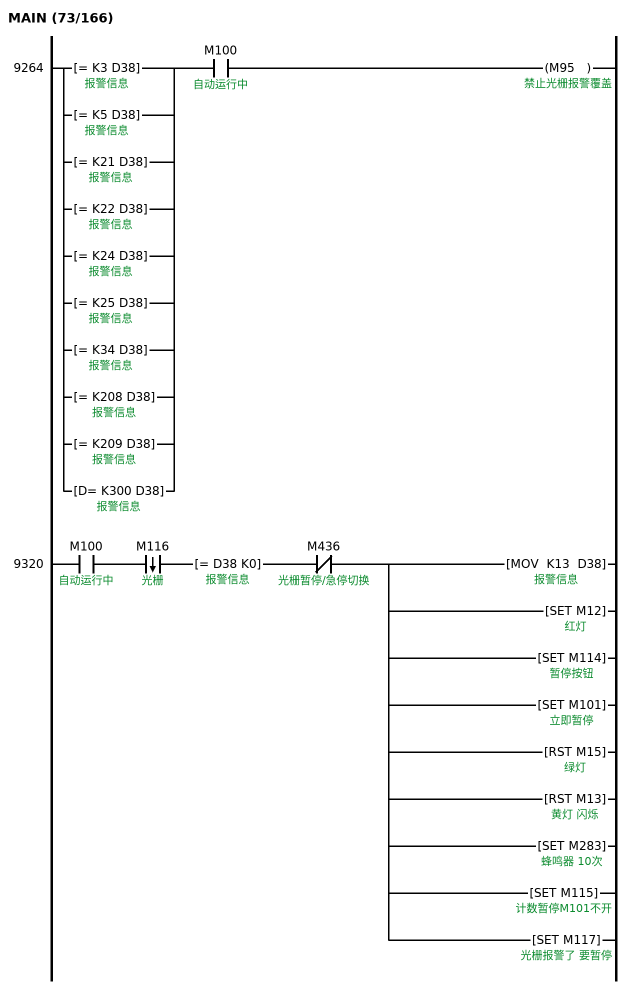
[picture p72: ladder of MAIN, rungs at steps 9264 to 9320]
9264  LD=     K3 D38  ; 报警信息
      OR=     K5 D38  ; 报警信息
      OR=     K21 D38  ; 报警信息
      OR=     K22 D38  ; 报警信息
      OR=     K24 D38  ; 报警信息
      OR=     K25 D38  ; 报警信息
      OR=     K34 D38  ; 报警信息
      OR=     K208 D38  ; 报警信息
      OR=     K209 D38  ; 报警信息
      ORD=    K300 D38  ; 报警信息
      AND     M100  ; 自动运行中
      OUT     M95  ; 禁止光栅报警覆盖
9320  LD      M100  ; 自动运行中
      ANDF    M116  ; 光栅
      AND=    D38 K0  ; 报警信息
      ANI     M436  ; 光栅暂停/急停切换
      MOV     K13 D38
      SET     M12  ; 红灯
      SET     M114  ; 暂停按钮
      SET     M101  ; 立即暂停
      RST     M15  ; 绿灯
      RST     M13  ; 黄灯 闪烁
      SET     M283  ; 蜂鸣器 10次
      SET     M115  ; 计数暂停M101不开
      SET     M117  ; 光栅报警了 要暂停
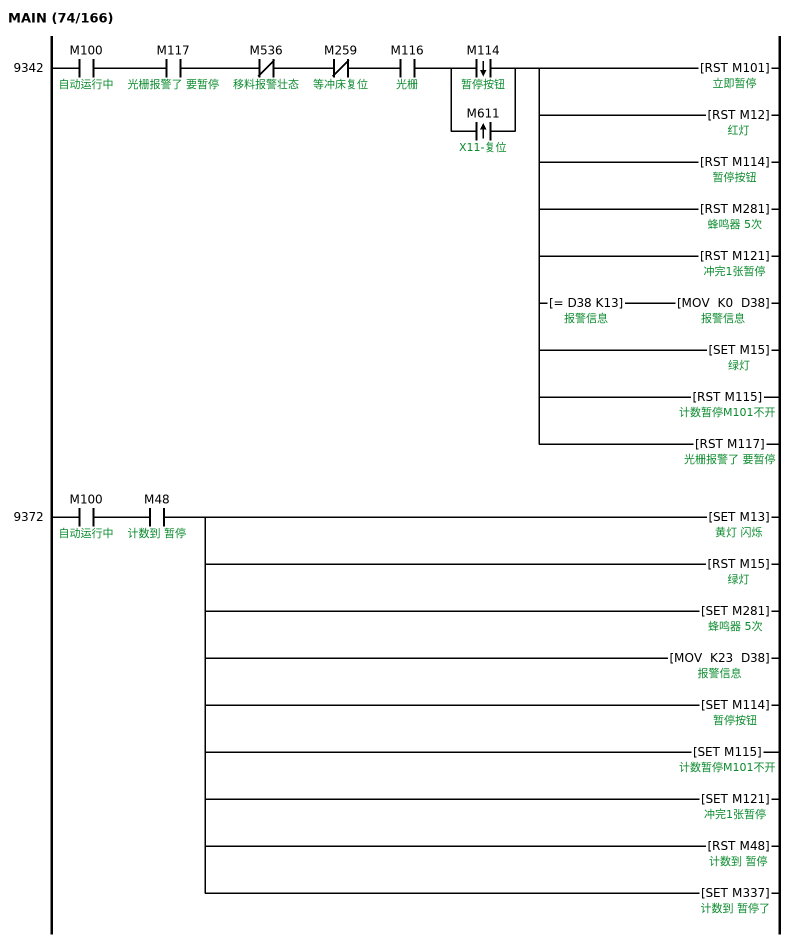
9342  LD      M100  ; 自动运行中
      AND     M117  ; 光栅报警了 要暂停
      ANI     M536  ; 移料报警壮态
      ANI     M259  ; 等冲床复位
      AND     M116  ; 光栅
      LDF     M114  ; 暂停按钮
      ORP     M611  ; X11-复位
      ANB
      RST     M101  ; 立即暂停
      RST     M12  ; 红灯
      RST     M114  ; 暂停按钮
      RST     M281  ; 蜂鸣器 5次
      RST     M121  ; 冲完1张暂停
      MPS
      AND=    D38 K13  ; 报警信息
      MOV     K0 D38
      MPP
      SET     M15  ; 绿灯
      RST     M115  ; 计数暂停M101不开
      RST     M117  ; 光栅报警了 要暂停
9372  LD      M100  ; 自动运行中
      AND     M48  ; 计数到 暂停
      SET     M13  ; 黄灯 闪烁
      RST     M15  ; 绿灯
      SET     M281  ; 蜂鸣器 5次
      MOV     K23 D38
      SET     M114  ; 暂停按钮
      SET     M115  ; 计数暂停M101不开
      SET     M121  ; 冲完1张暂停
      RST     M48  ; 计数到 暂停
      SET     M337  ; 计数到 暂停了
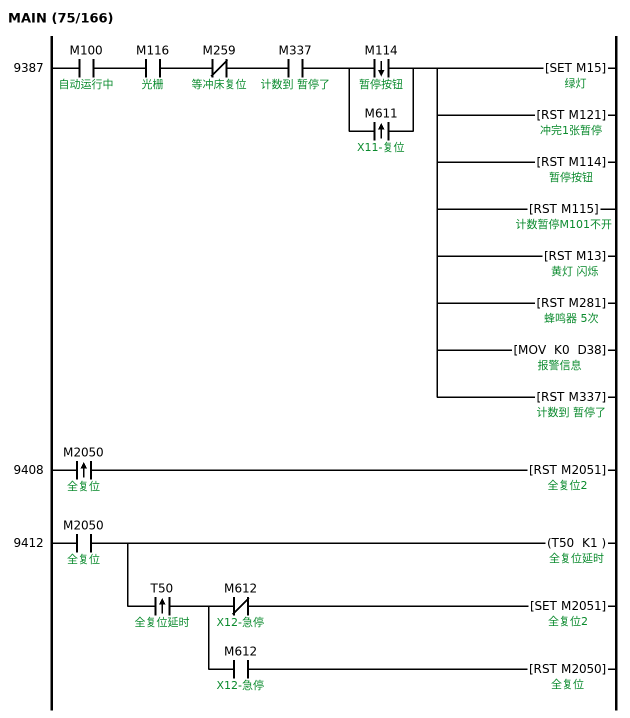
9387  LD      M100  ; 自动运行中
      AND     M116  ; 光栅
      ANI     M259  ; 等冲床复位
      AND     M337  ; 计数到 暂停了
      LDF     M114  ; 暂停按钮
      ORP     M611  ; X11-复位
      ANB
      SET     M15  ; 绿灯
      RST     M121  ; 冲完1张暂停
      RST     M114  ; 暂停按钮
      RST     M115  ; 计数暂停M101不开
      RST     M13  ; 黄灯 闪烁
      RST     M281  ; 蜂鸣器 5次
      MOV     K0 D38
      RST     M337  ; 计数到 暂停了
9408  LDP     M2050  ; 全复位
      RST     M2051  ; 全复位2
9412  LD      M2050  ; 全复位
      OUT     T50 K1  ; 全复位延时
      ANDP    T50  ; 全复位延时
      MPS
      ANI     M612  ; X12-急停
      SET     M2051  ; 全复位2
      MPP
      AND     M612  ; X12-急停
      RST     M2050  ; 全复位
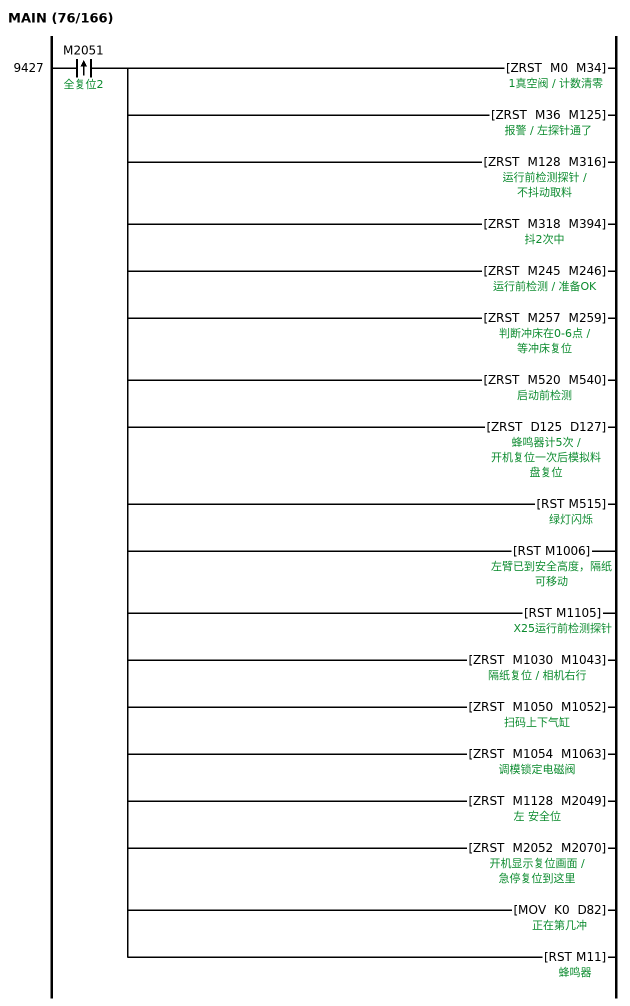
9427  LDP     M2051  ; 全复位2
      ZRST    M0 M34
      ZRST    M36 M125
      ZRST    M128 M316
      ZRST    M318 M394
      ZRST    M245 M246
      ZRST    M257 M259
      ZRST    M520 M540
      ZRST    D125 D127
      RST     M515  ; 绿灯闪烁
      RST     M1006  ; 左臂已到安全高度，隔纸可移动
      RST     M1105  ; X25运行前检测探针
      ZRST    M1030 M1043
      ZRST    M1050 M1052
      ZRST    M1054 M1063
      ZRST    M1128 M2049
      ZRST    M2052 M2070
      MOV     K0 D82
      RST     M11  ; 蜂鸣器
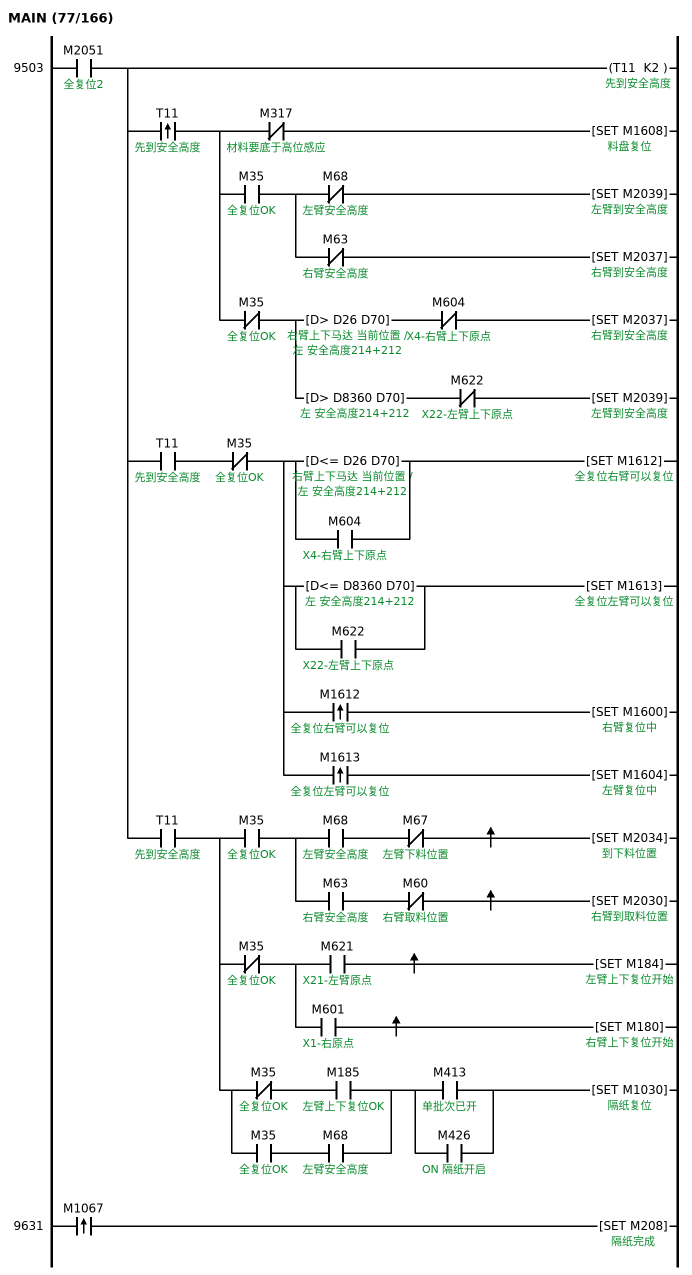
9503  LD      M2051  ; 全复位2
      OUT     T11 K2  ; 先到安全高度
      MPS
      ANDP    T11  ; 先到安全高度
      MPS
      ANI     M317  ; 材料要底于高位感应
      SET     M1608  ; 料盘复位
      MRD
      AND     M35  ; 全复位OK
      MPS
      ANI     M68  ; 左臂安全高度
      SET     M2039  ; 左臂到安全高度
      MPP
      ANI     M63  ; 右臂安全高度
      SET     M2037  ; 右臂到安全高度
      MPP
      ANI     M35  ; 全复位OK
      MPS
      ANDD>   D26 D70  ; 右臂上下马达 当前位置 / 左 安全高度214+212
      ANI     M604  ; X4-右臂上下原点
      SET     M2037  ; 右臂到安全高度
      MPP
      ANDD>   D8360 D70  ; 左 安全高度214+212
      ANI     M622  ; X22-左臂上下原点
      SET     M2039  ; 左臂到安全高度
      MRD
      AND     T11  ; 先到安全高度
      ANI     M35  ; 全复位OK
      MPS
      LDD<=   D26 D70  ; 右臂上下马达 当前位置 / 左 安全高度214+212
      OR      M604  ; X4-右臂上下原点
      ANB
      SET     M1612  ; 全复位右臂可以复位
      MRD
      LDD<=   D8360 D70  ; 左 安全高度214+212
      OR      M622  ; X22-左臂上下原点
      ANB
      SET     M1613  ; 全复位左臂可以复位
      MRD
      ANDP    M1612  ; 全复位右臂可以复位
      SET     M1600  ; 右臂复位中
      MPP
      ANDP    M1613  ; 全复位左臂可以复位
      SET     M1604  ; 左臂复位中
      MPP
      AND     T11  ; 先到安全高度
      MPS
      AND     M35  ; 全复位OK
      MPS
      AND     M68  ; 左臂安全高度
      ANI     M67  ; 左臂下料位置
      MEP
      SET     M2034  ; 到下料位置
      MPP
      AND     M63  ; 右臂安全高度
      ANI     M60  ; 右臂取料位置
      MEP
      SET     M2030  ; 右臂到取料位置
      MRD
      ANI     M35  ; 全复位OK
      MPS
      AND     M621  ; X21-左臂原点
      MEP
      SET     M184  ; 左臂上下复位开始
      MPP
      AND     M601  ; X1-右原点
      MEP
      SET     M180  ; 右臂上下复位开始
      MPP
      LDI     M35  ; 全复位OK
      AND     M185  ; 左臂上下复位OK
      LD      M35  ; 全复位OK
      AND     M68  ; 左臂安全高度
      ORB
      ANB
      LD      M413  ; 单批次已开
      OR      M426  ; ON 隔纸开启
      ANB
      SET     M1030  ; 隔纸复位
9631  LDP     M1067
      SET     M208  ; 隔纸完成
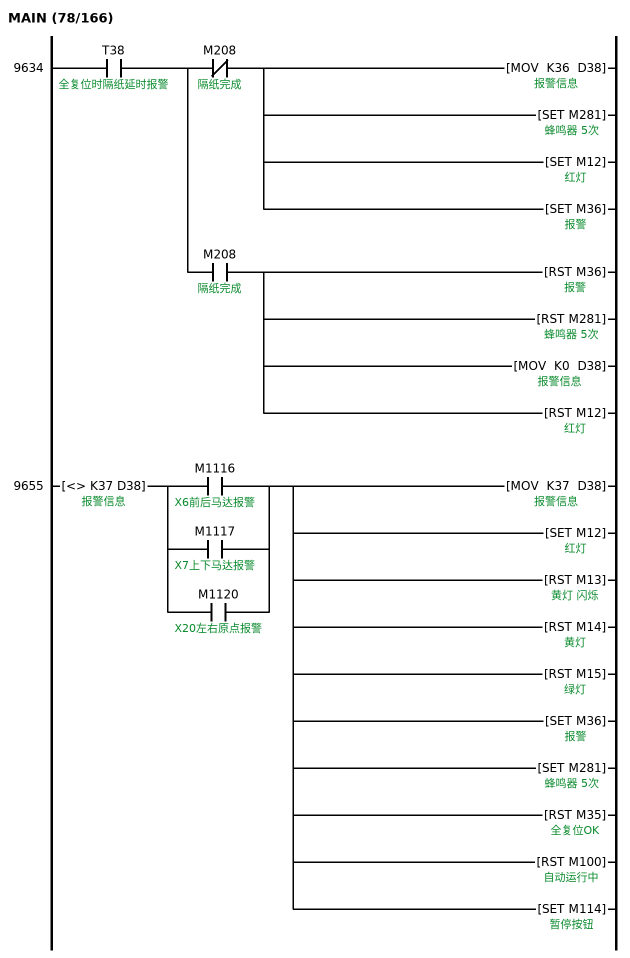
9634  LD      T38  ; 全复位时隔纸延时报警
      MPS
      ANI     M208  ; 隔纸完成
      MOV     K36 D38
      SET     M281  ; 蜂鸣器 5次
      SET     M12  ; 红灯
      SET     M36  ; 报警
      MPP
      AND     M208  ; 隔纸完成
      RST     M36  ; 报警
      RST     M281  ; 蜂鸣器 5次
      MOV     K0 D38
      RST     M12  ; 红灯
9655  LD<>    K37 D38  ; 报警信息
      LD      M1116  ; X6前后马达报警
      OR      M1117  ; X7上下马达报警
      OR      M1120  ; X20左右原点报警
      ANB
      MOV     K37 D38
      SET     M12  ; 红灯
      RST     M13  ; 黄灯 闪烁
      RST     M14  ; 黄灯
      RST     M15  ; 绿灯
      SET     M36  ; 报警
      SET     M281  ; 蜂鸣器 5次
      RST     M35  ; 全复位OK
      RST     M100  ; 自动运行中
      SET     M114  ; 暂停按钮
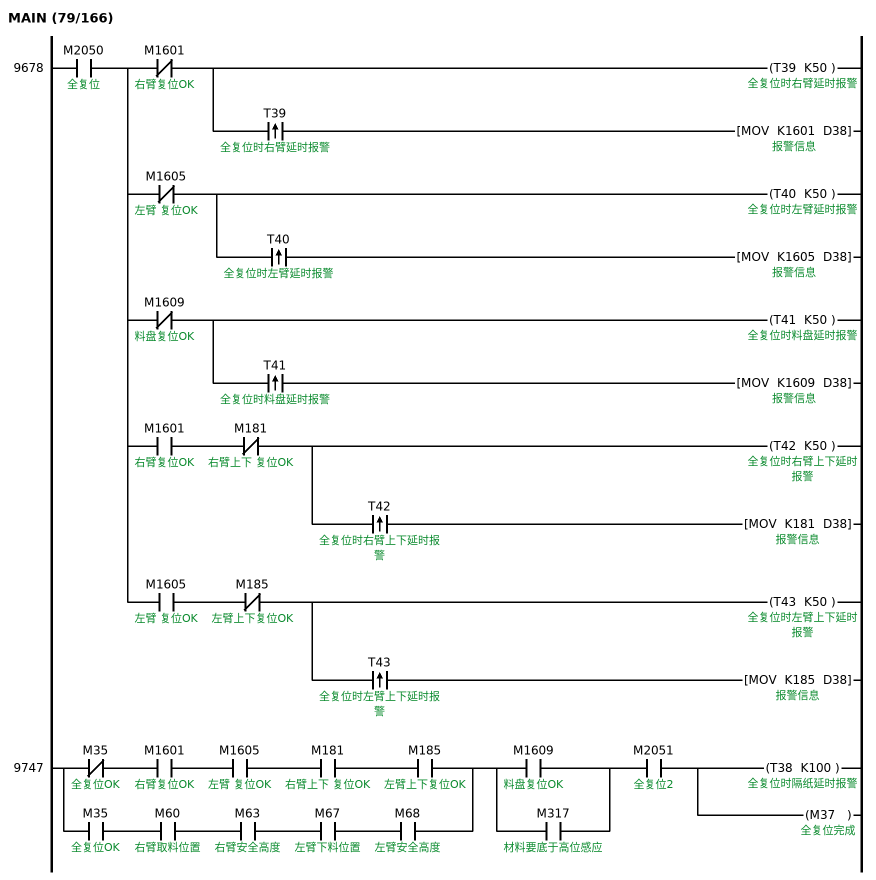
9678  LD      M2050  ; 全复位
      MPS
      ANI     M1601  ; 右臂复位OK
      OUT     T39 K50  ; 全复位时右臂延时报警
      ANDP    T39  ; 全复位时右臂延时报警
      MOV     K1601 D38
      MRD
      ANI     M1605  ; 左臂 复位OK
      OUT     T40 K50  ; 全复位时左臂延时报警
      ANDP    T40  ; 全复位时左臂延时报警
      MOV     K1605 D38
      MRD
      ANI     M1609  ; 料盘复位OK
      OUT     T41 K50  ; 全复位时料盘延时报警
      ANDP    T41  ; 全复位时料盘延时报警
      MOV     K1609 D38
      MRD
      AND     M1601  ; 右臂复位OK
      ANI     M181  ; 右臂上下 复位OK
      OUT     T42 K50  ; 全复位时右臂上下延时报警
      ANDP    T42  ; 全复位时右臂上下延时报警
      MOV     K181 D38
      MPP
      AND     M1605  ; 左臂 复位OK
      ANI     M185  ; 左臂上下复位OK
      OUT     T43 K50  ; 全复位时左臂上下延时报警
      ANDP    T43  ; 全复位时左臂上下延时报警
      MOV     K185 D38
9747  LDI     M35  ; 全复位OK
      AND     M1601  ; 右臂复位OK
      AND     M1605  ; 左臂 复位OK
      AND     M181  ; 右臂上下 复位OK
      AND     M185  ; 左臂上下复位OK
      LD      M35  ; 全复位OK
      AND     M60  ; 右臂取料位置
      AND     M63  ; 右臂安全高度
      AND     M67  ; 左臂下料位置
      AND     M68  ; 左臂安全高度
      ORB
      LD      M1609  ; 料盘复位OK
      OR      M317  ; 材料要底于高位感应
      ANB
      AND     M2051  ; 全复位2
      OUT     T38 K100  ; 全复位时隔纸延时报警
      OUT     M37  ; 全复位完成
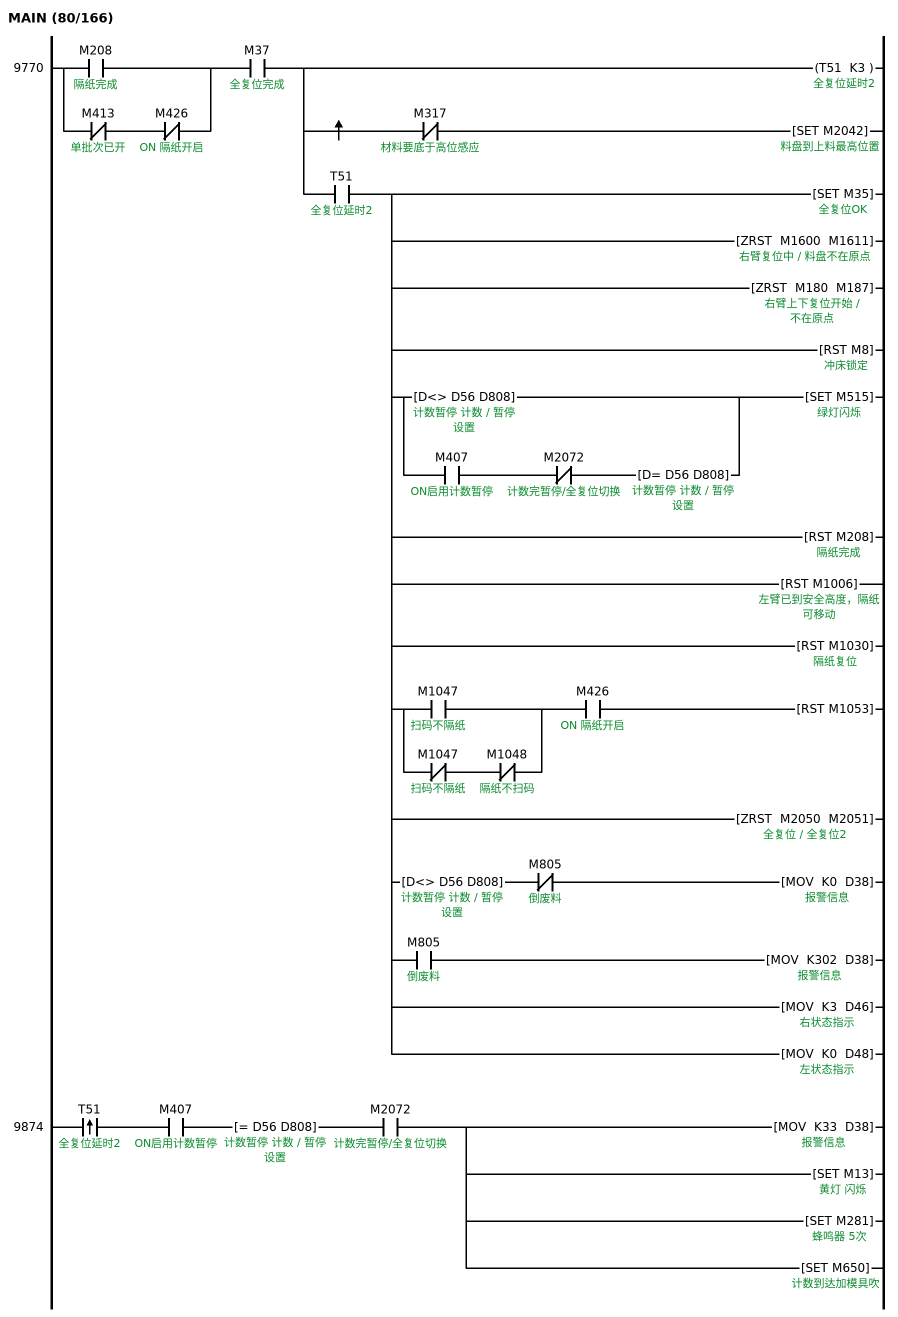
9770  LD      M208  ; 隔纸完成
      LDI     M413  ; 单批次已开
      ANI     M426  ; ON 隔纸开启
      ORB
      AND     M37  ; 全复位完成
      OUT     T51 K3  ; 全复位延时2
      MPS
      MEP
      ANI     M317  ; 材料要底于高位感应
      SET     M2042  ; 料盘到上料最高位置
      MPP
      AND     T51  ; 全复位延时2
      SET     M35  ; 全复位OK
      ZRST    M1600 M1611
      ZRST    M180 M187  ; 不在原点
      RST     M8  ; 冲床锁定
      MPS
      LDD<>   D56 D808  ; 计数暂停 计数 / 暂停 设置
      LD      M407  ; ON启用计数暂停
      ANI     M2072  ; 计数完暂停/全复位切换
      ANDD=   D56 D808  ; 计数暂停 计数 / 暂停 设置
      ORB
      ANB
      SET     M515  ; 绿灯闪烁
      MPP
      RST     M208  ; 隔纸完成
      RST     M1006  ; 左臂已到安全高度，隔纸可移动
      RST     M1030  ; 隔纸复位
      MPS
      LD      M1047  ; 扫码不隔纸
      LDI     M1047  ; 扫码不隔纸
      ANI     M1048  ; 隔纸不扫码
      ORB
      ANB
      AND     M426  ; ON 隔纸开启
      RST     M1053
      MPP
      ZRST    M2050 M2051
      MPS
      ANDD<>  D56 D808  ; 计数暂停 计数 / 暂停 设置
      ANI     M805  ; 倒废料
      MOV     K0 D38
      MRD
      AND     M805  ; 倒废料
      MOV     K302 D38
      MPP
      MOV     K3 D46
      MOV     K0 D48
9874  LDP     T51  ; 全复位延时2
      AND     M407  ; ON启用计数暂停
      AND=    D56 D808  ; 计数暂停 计数 / 暂停 设置
      AND     M2072  ; 计数完暂停/全复位切换
      MOV     K33 D38
      SET     M13  ; 黄灯 闪烁
      SET     M281  ; 蜂鸣器 5次
      SET     M650  ; 计数到达加模具吹
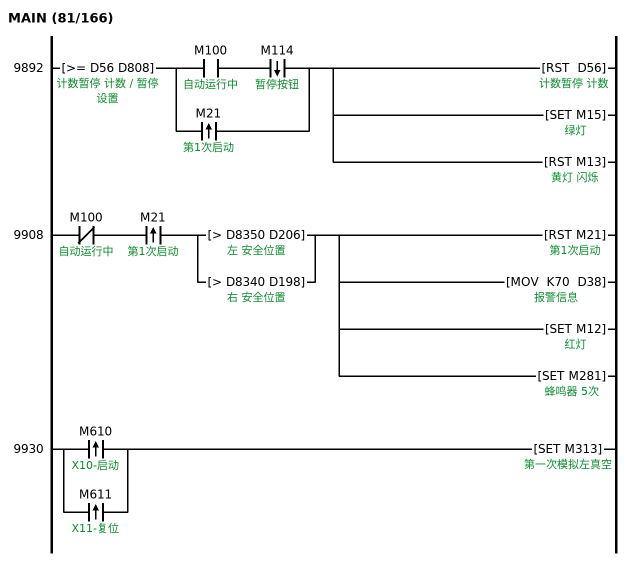
9892  LD>=    D56 D808  ; 计数暂停 计数 / 暂停 设置
      LD      M100  ; 自动运行中
      ANDF    M114  ; 暂停按钮
      ORP     M21  ; 第1次启动
      ANB
      RST     D56  ; 计数暂停 计数
      SET     M15  ; 绿灯
      RST     M13  ; 黄灯 闪烁
9908  LDI     M100  ; 自动运行中
      ANDP    M21  ; 第1次启动
      LD>     D8350 D206  ; 左 安全位置
      OR>     D8340 D198  ; 右 安全位置
      ANB
      RST     M21  ; 第1次启动
      MOV     K70 D38
      SET     M12  ; 红灯
      SET     M281  ; 蜂鸣器 5次
9930  LDP     M610  ; X10-启动
      ORP     M611  ; X11-复位
      SET     M313  ; 第一次模拟左真空
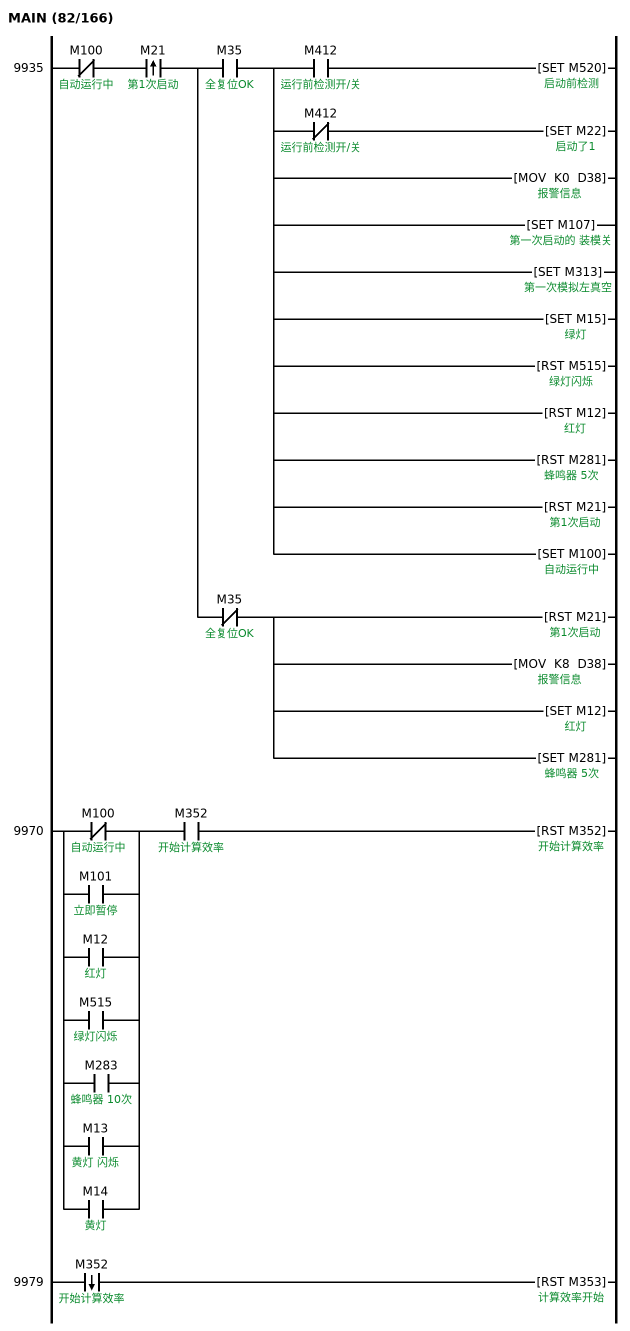
9935  LDI     M100  ; 自动运行中
      ANDP    M21  ; 第1次启动
      MPS
      AND     M35  ; 全复位OK
      MPS
      AND     M412  ; 运行前检测开/关
      SET     M520  ; 启动前检测
      MRD
      ANI     M412  ; 运行前检测开/关
      SET     M22  ; 启动了1
      MPP
      MOV     K0 D38
      SET     M107  ; 第一次启动的 装模关
      SET     M313  ; 第一次模拟左真空
      SET     M15  ; 绿灯
      RST     M515  ; 绿灯闪烁
      RST     M12  ; 红灯
      RST     M281  ; 蜂鸣器 5次
      RST     M21  ; 第1次启动
      SET     M100  ; 自动运行中
      MPP
      ANI     M35  ; 全复位OK
      RST     M21  ; 第1次启动
      MOV     K8 D38
      SET     M12  ; 红灯
      SET     M281  ; 蜂鸣器 5次
9970  LDI     M100  ; 自动运行中
      OR      M101  ; 立即暂停
      OR      M12  ; 红灯
      OR      M515  ; 绿灯闪烁
      OR      M283  ; 蜂鸣器 10次
      OR      M13  ; 黄灯 闪烁
      OR      M14  ; 黄灯
      AND     M352  ; 开始计算效率
      RST     M352  ; 开始计算效率
9979  LDF     M352  ; 开始计算效率
      RST     M353  ; 计算效率开始
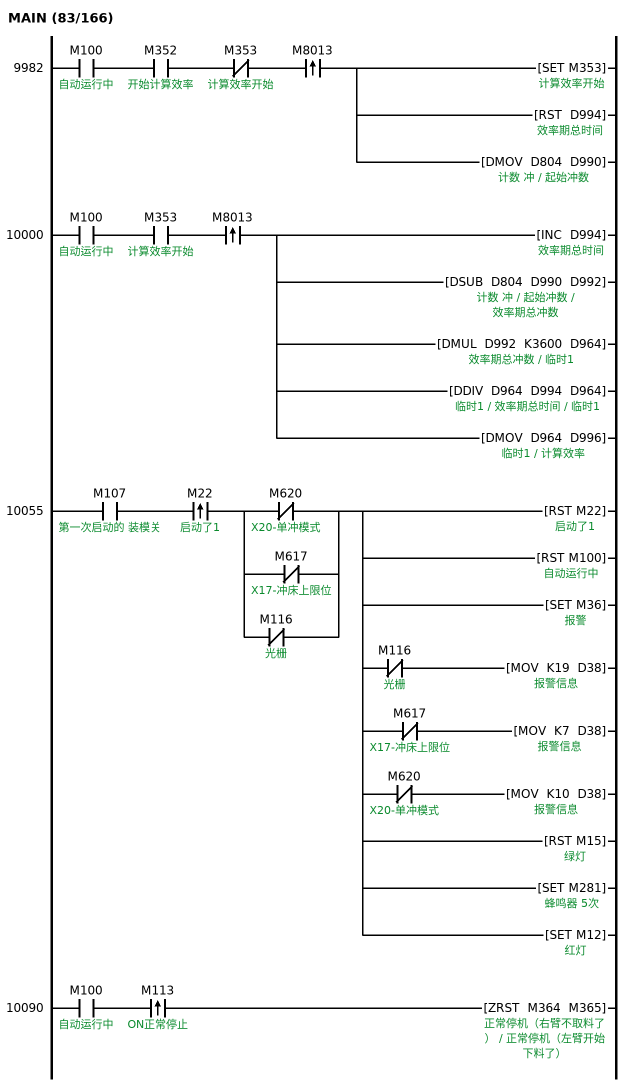
9982  LD      M100  ; 自动运行中
      AND     M352  ; 开始计算效率
      ANI     M353  ; 计算效率开始
      ANDP    M8013
      SET     M353  ; 计算效率开始
      RST     D994  ; 效率期总时间
      DMOV    D804 D990  ; 起始冲数
10000 LD      M100  ; 自动运行中
      AND     M353  ; 计算效率开始
      ANDP    M8013
      INC     D994
      DSUB    D804 D990 D992
      DMUL    D992 K3600 D964
      DDIV    D964 D994 D964
      DMOV    D964 D996
10055 LD      M107  ; 第一次启动的 装模关
      ANDP    M22  ; 启动了1
      LDI     M620  ; X20-单冲模式
      ORI     M617  ; X17-冲床上限位
      ORI     M116  ; 光栅
      ANB
      RST     M22  ; 启动了1
      RST     M100  ; 自动运行中
      SET     M36  ; 报警
      MPS
      ANI     M116  ; 光栅
      MOV     K19 D38
      MRD
      ANI     M617  ; X17-冲床上限位
      MOV     K7 D38
      MRD
      ANI     M620  ; X20-单冲模式
      MOV     K10 D38
      MPP
      RST     M15  ; 绿灯
      SET     M281  ; 蜂鸣器 5次
      SET     M12  ; 红灯
10090 LD      M100  ; 自动运行中
      ANDP    M113  ; ON正常停止
      ZRST    M364 M365  ; 正常停机（右臂不取料了） / 正常停机（左臂开始下料了）
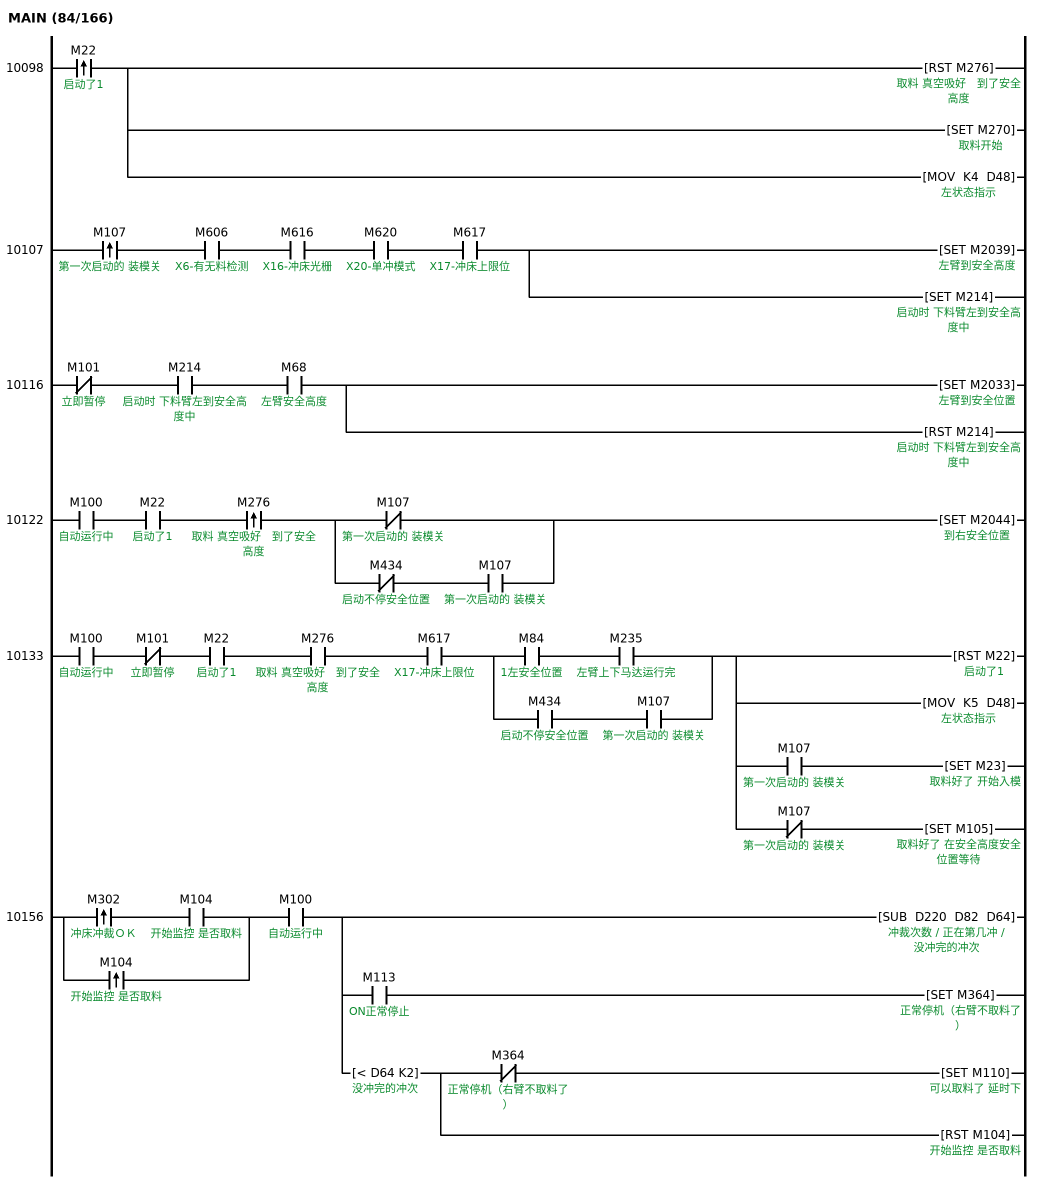
10098 LDP     M22  ; 启动了1
      RST     M276  ; 取料 真空吸好　到了安全高度
      SET     M270  ; 取料开始
      MOV     K4 D48
10107 LDP     M107  ; 第一次启动的 装模关
      AND     M606  ; X6-有无料检测
      AND     M616  ; X16-冲床光栅
      AND     M620  ; X20-单冲模式
      AND     M617  ; X17-冲床上限位
      SET     M2039  ; 左臂到安全高度
      SET     M214  ; 启动时 下料臂左到安全高度中
10116 LDI     M101  ; 立即暂停
      AND     M214  ; 启动时 下料臂左到安全高度中
      AND     M68  ; 左臂安全高度
      SET     M2033  ; 左臂到安全位置
      RST     M214  ; 启动时 下料臂左到安全高度中
10122 LD      M100  ; 自动运行中
      AND     M22  ; 启动了1
      ANDP    M276  ; 取料 真空吸好　到了安全高度
      LDI     M107  ; 第一次启动的 装模关
      LDI     M434  ; 启动不停安全位置
      AND     M107  ; 第一次启动的 装模关
      ORB
      ANB
      SET     M2044  ; 到右安全位置
10133 LD      M100  ; 自动运行中
      ANI     M101  ; 立即暂停
      AND     M22  ; 启动了1
      AND     M276  ; 取料 真空吸好　到了安全高度
      AND     M617  ; X17-冲床上限位
      LD      M84  ; 1左安全位置
      AND     M235  ; 左臂上下马达运行完
      LD      M434  ; 启动不停安全位置
      AND     M107  ; 第一次启动的 装模关
      ORB
      ANB
      RST     M22  ; 启动了1
      MOV     K5 D48
      MPS
      AND     M107  ; 第一次启动的 装模关
      SET     M23  ; 取料好了 开始入模
      MPP
      ANI     M107  ; 第一次启动的 装模关
      SET     M105  ; 取料好了 在安全高度安全位置等待
10156 LDP     M302  ; 冲床冲裁ＯＫ
      AND     M104  ; 开始监控 是否取料
      ORP     M104  ; 开始监控 是否取料
      AND     M100  ; 自动运行中
      SUB     D220 D82 D64  ; 没冲完的冲次
      MPS
      AND     M113  ; ON正常停止
      SET     M364  ; 正常停机（右臂不取料了）
      MPP
      AND<    D64 K2  ; 没冲完的冲次
      MPS
      ANI     M364  ; 正常停机（右臂不取料了）
      SET     M110  ; 可以取料了 延时下
      MPP
      RST     M104  ; 开始监控 是否取料
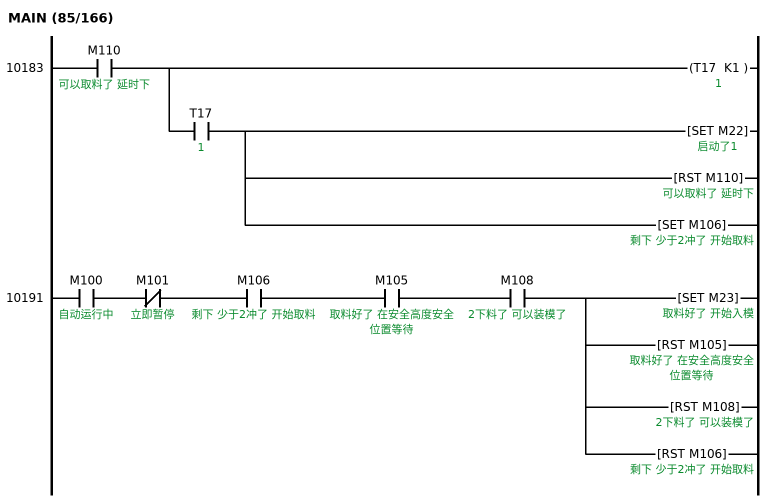
10183 LD      M110  ; 可以取料了 延时下
      OUT     T17 K1  ; 1
      AND     T17  ; 1
      SET     M22  ; 启动了1
      RST     M110  ; 可以取料了 延时下
      SET     M106  ; 剩下 少于2冲了 开始取料
10191 LD      M100  ; 自动运行中
      ANI     M101  ; 立即暂停
      AND     M106  ; 剩下 少于2冲了 开始取料
      AND     M105  ; 取料好了 在安全高度安全位置等待
      AND     M108  ; 2下料了 可以装模了
      SET     M23  ; 取料好了 开始入模
      RST     M105  ; 取料好了 在安全高度安全位置等待
      RST     M108  ; 2下料了 可以装模了
      RST     M106  ; 剩下 少于2冲了 开始取料
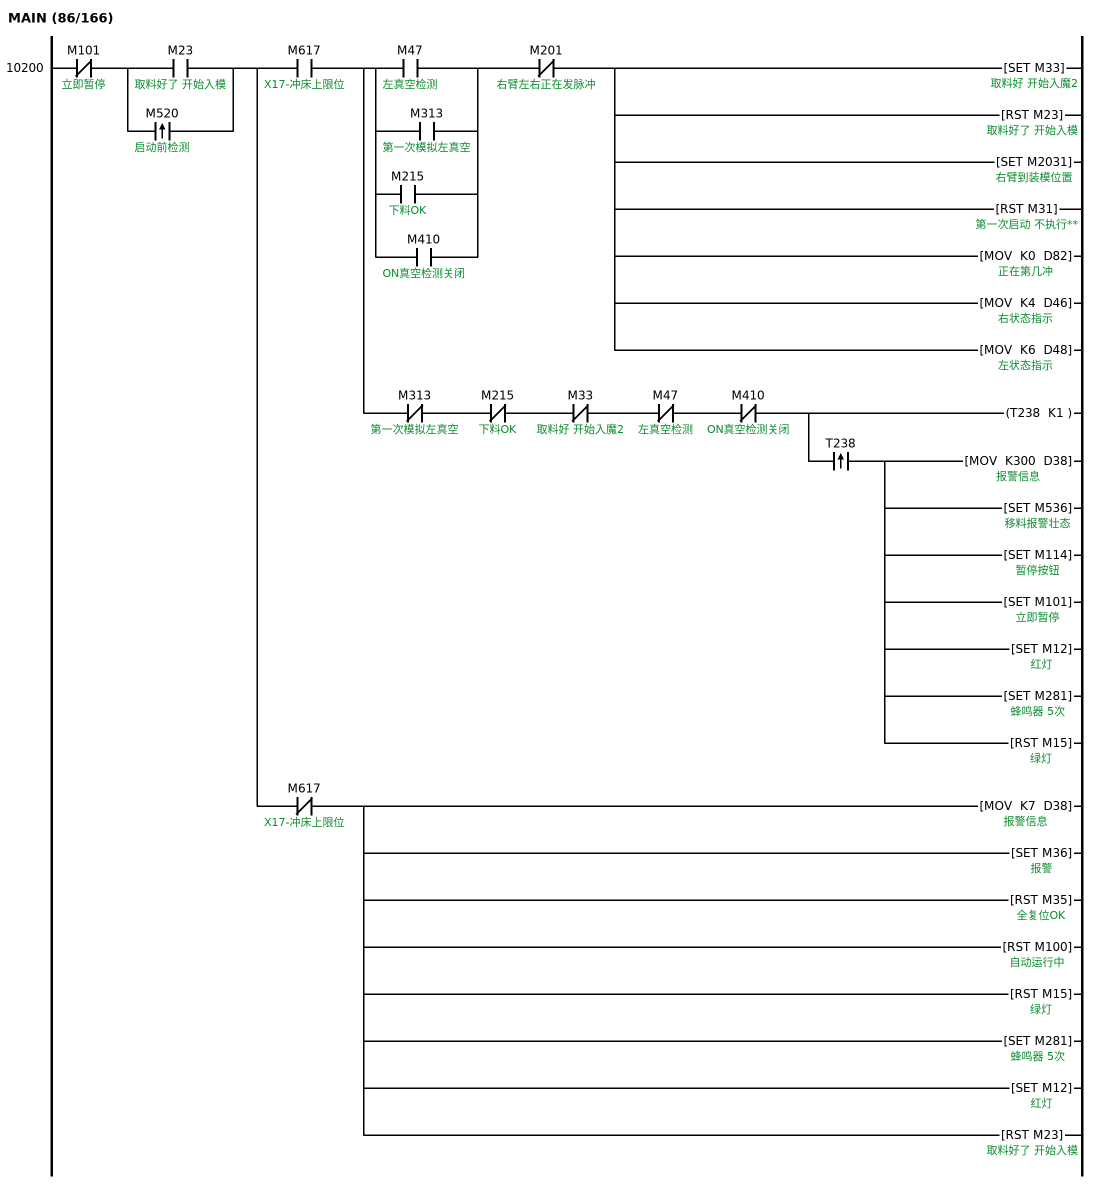
10200 LDI     M101  ; 立即暂停
      LD      M23  ; 取料好了 开始入模
      ORP     M520  ; 启动前检测
      ANB
      MPS
      AND     M617  ; X17-冲床上限位
      MPS
      LD      M47  ; 左真空检测
      OR      M313  ; 第一次模拟左真空
      OR      M215  ; 下料OK
      OR      M410  ; ON真空检测关闭
      ANB
      ANI     M201  ; 右臂左右正在发脉冲
      SET     M33  ; 取料好 开始入魔2
      RST     M23  ; 取料好了 开始入模
      SET     M2031  ; 右臂到装模位置
      RST     M31  ; 第一次启动 不执行**
      MOV     K0 D82
      MOV     K4 D46
      MOV     K6 D48
      MPP
      ANI     M313  ; 第一次模拟左真空
      ANI     M215  ; 下料OK
      ANI     M33  ; 取料好 开始入魔2
      ANI     M47  ; 左真空检测
      ANI     M410  ; ON真空检测关闭
      OUT     T238 K1
      ANDP    T238
      MOV     K300 D38
      SET     M536  ; 移料报警壮态
      SET     M114  ; 暂停按钮
      SET     M101  ; 立即暂停
      SET     M12  ; 红灯
      SET     M281  ; 蜂鸣器 5次
      RST     M15  ; 绿灯
      MPP
      ANI     M617  ; X17-冲床上限位
      MOV     K7 D38
      SET     M36  ; 报警
      RST     M35  ; 全复位OK
      RST     M100  ; 自动运行中
      RST     M15  ; 绿灯
      SET     M281  ; 蜂鸣器 5次
      SET     M12  ; 红灯
      RST     M23  ; 取料好了 开始入模
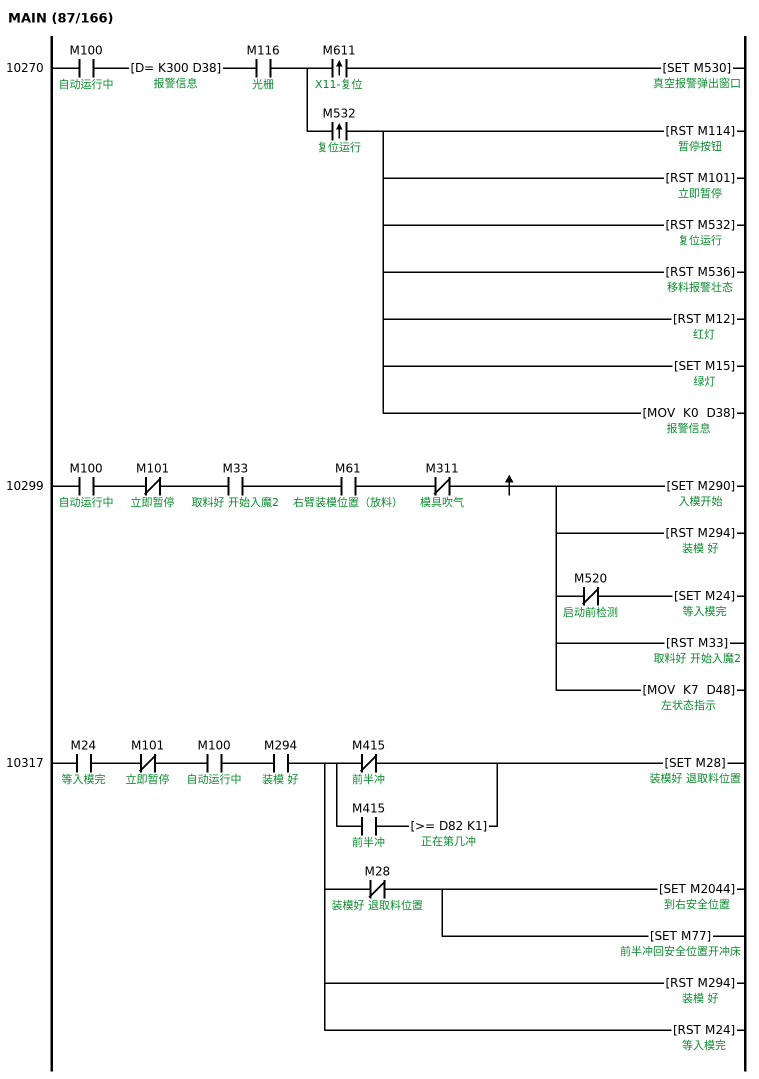
10270 LD      M100  ; 自动运行中
      ANDD=   K300 D38  ; 报警信息
      AND     M116  ; 光栅
      MPS
      ANDP    M611  ; X11-复位
      SET     M530  ; 真空报警弹出窗口
      MPP
      ANDP    M532  ; 复位运行
      RST     M114  ; 暂停按钮
      RST     M101  ; 立即暂停
      RST     M532  ; 复位运行
      RST     M536  ; 移料报警壮态
      RST     M12  ; 红灯
      SET     M15  ; 绿灯
      MOV     K0 D38
10299 LD      M100  ; 自动运行中
      ANI     M101  ; 立即暂停
      AND     M33  ; 取料好 开始入魔2
      AND     M61  ; 右臂装模位置（放料）
      ANI     M311  ; 模具吹气
      MEP
      SET     M290  ; 入模开始
      RST     M294  ; 装模 好
      MPS
      ANI     M520  ; 启动前检测
      SET     M24  ; 等入模完
      MPP
      RST     M33  ; 取料好 开始入魔2
      MOV     K7 D48
10317 LD      M24  ; 等入模完
      ANI     M101  ; 立即暂停
      AND     M100  ; 自动运行中
      AND     M294  ; 装模 好
      MPS
      LDI     M415  ; 前半冲
      LD      M415  ; 前半冲
      AND>=   D82 K1  ; 正在第几冲
      ORB
      ANB
      SET     M28  ; 装模好 退取料位置
      MRD
      ANI     M28  ; 装模好 退取料位置
      SET     M2044  ; 到右安全位置
      SET     M77  ; 前半冲回安全位置开冲床
      MPP
      RST     M294  ; 装模 好
      RST     M24  ; 等入模完
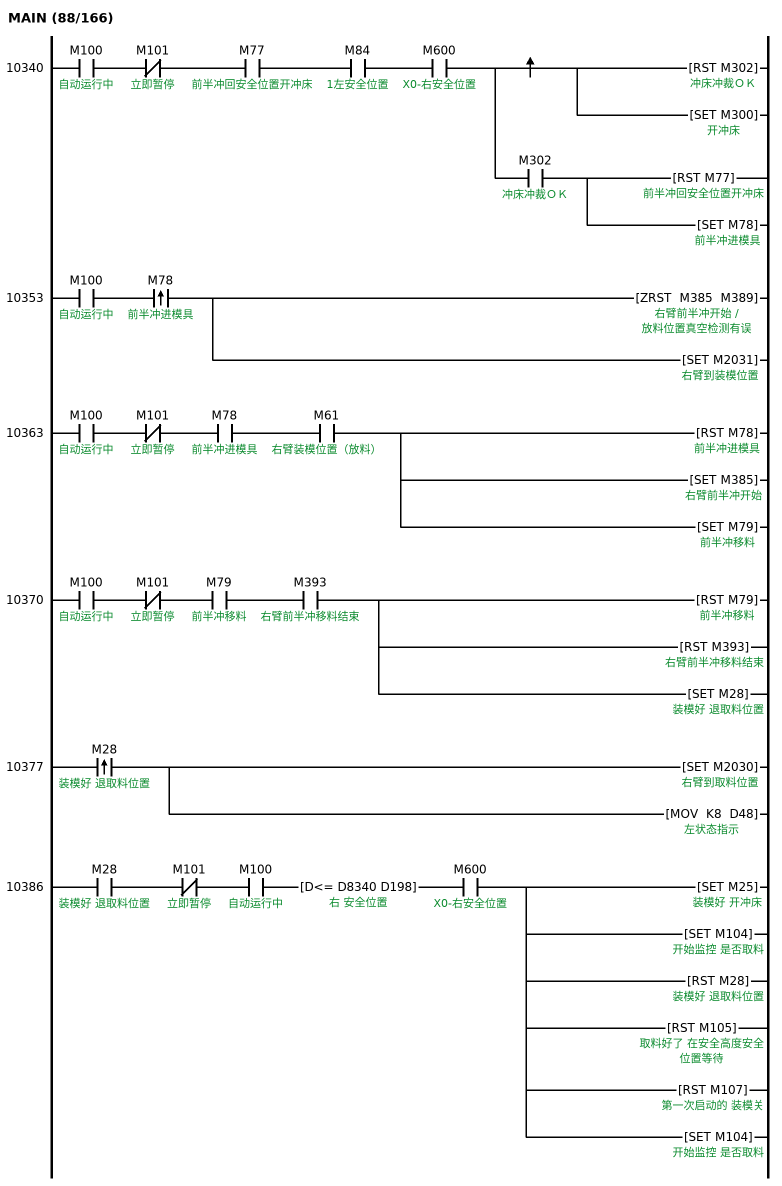
10340 LD      M100  ; 自动运行中
      ANI     M101  ; 立即暂停
      AND     M77  ; 前半冲回安全位置开冲床
      AND     M84  ; 1左安全位置
      AND     M600  ; X0-右安全位置
      MPS
      MEP
      RST     M302  ; 冲床冲裁ＯＫ
      SET     M300  ; 开冲床
      MPP
      AND     M302  ; 冲床冲裁ＯＫ
      RST     M77  ; 前半冲回安全位置开冲床
      SET     M78  ; 前半冲进模具
10353 LD      M100  ; 自动运行中
      ANDP    M78  ; 前半冲进模具
      ZRST    M385 M389  ; 右臂前半冲开始 / 放料位置真空检测有误
      SET     M2031  ; 右臂到装模位置
10363 LD      M100  ; 自动运行中
      ANI     M101  ; 立即暂停
      AND     M78  ; 前半冲进模具
      AND     M61  ; 右臂装模位置（放料）
      RST     M78  ; 前半冲进模具
      SET     M385  ; 右臂前半冲开始
      SET     M79  ; 前半冲移料
10370 LD      M100  ; 自动运行中
      ANI     M101  ; 立即暂停
      AND     M79  ; 前半冲移料
      AND     M393  ; 右臂前半冲移料结束
      RST     M79  ; 前半冲移料
      RST     M393  ; 右臂前半冲移料结束
      SET     M28  ; 装模好 退取料位置
10377 LDP     M28  ; 装模好 退取料位置
      SET     M2030  ; 右臂到取料位置
      MOV     K8 D48
10386 LD      M28  ; 装模好 退取料位置
      ANI     M101  ; 立即暂停
      AND     M100  ; 自动运行中
      ANDD<=  D8340 D198  ; 右 安全位置
      AND     M600  ; X0-右安全位置
      SET     M25  ; 装模好 开冲床
      SET     M104  ; 开始监控 是否取料
      RST     M28  ; 装模好 退取料位置
      RST     M105  ; 取料好了 在安全高度安全位置等待
      RST     M107  ; 第一次启动的 装模关
      SET     M104  ; 开始监控 是否取料
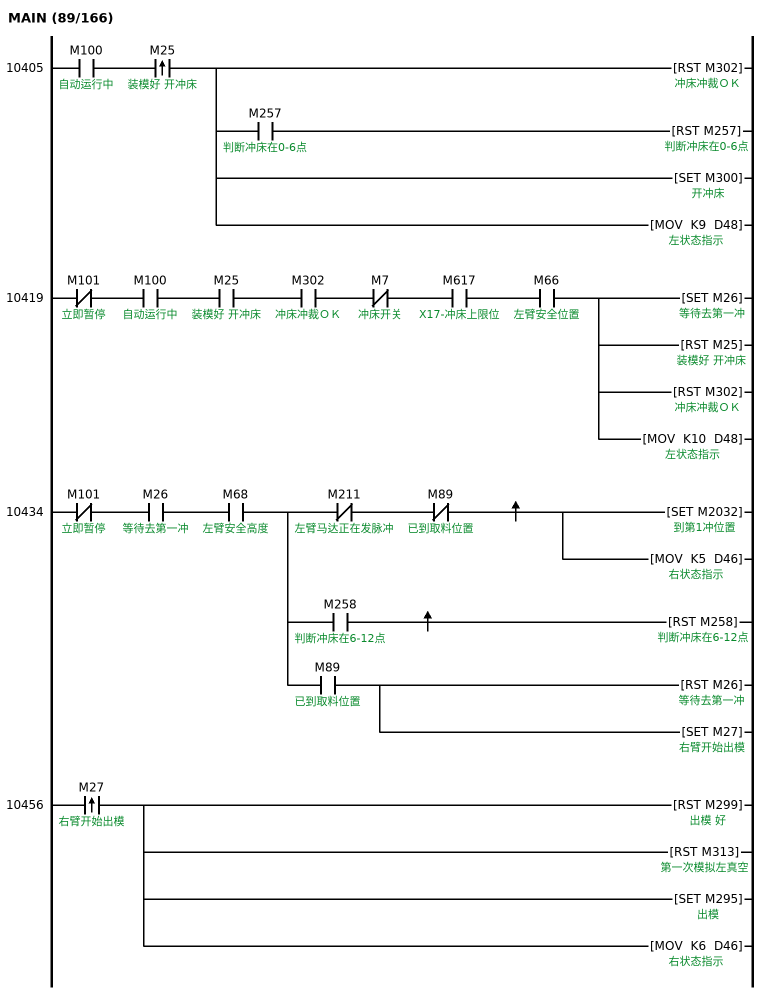
10405 LD      M100  ; 自动运行中
      ANDP    M25  ; 装模好 开冲床
      RST     M302  ; 冲床冲裁ＯＫ
      MPS
      AND     M257  ; 判断冲床在0-6点
      RST     M257  ; 判断冲床在0-6点
      MPP
      SET     M300  ; 开冲床
      MOV     K9 D48
10419 LDI     M101  ; 立即暂停
      AND     M100  ; 自动运行中
      AND     M25  ; 装模好 开冲床
      AND     M302  ; 冲床冲裁ＯＫ
      ANI     M7  ; 冲床开关
      AND     M617  ; X17-冲床上限位
      AND     M66  ; 左臂安全位置
      SET     M26  ; 等待去第一冲
      RST     M25  ; 装模好 开冲床
      RST     M302  ; 冲床冲裁ＯＫ
      MOV     K10 D48
10434 LDI     M101  ; 立即暂停
      AND     M26  ; 等待去第一冲
      AND     M68  ; 左臂安全高度
      MPS
      ANI     M211  ; 左臂马达正在发脉冲
      ANI     M89  ; 已到取料位置
      MEP
      SET     M2032  ; 到第1冲位置
      MOV     K5 D46
      MRD
      AND     M258  ; 判断冲床在6-12点
      MEP
      RST     M258  ; 判断冲床在6-12点
      MPP
      AND     M89  ; 已到取料位置
      RST     M26  ; 等待去第一冲
      SET     M27  ; 右臂开始出模
10456 LDP     M27  ; 右臂开始出模
      RST     M299  ; 出模 好
      RST     M313  ; 第一次模拟左真空
      SET     M295  ; 出模
      MOV     K6 D46
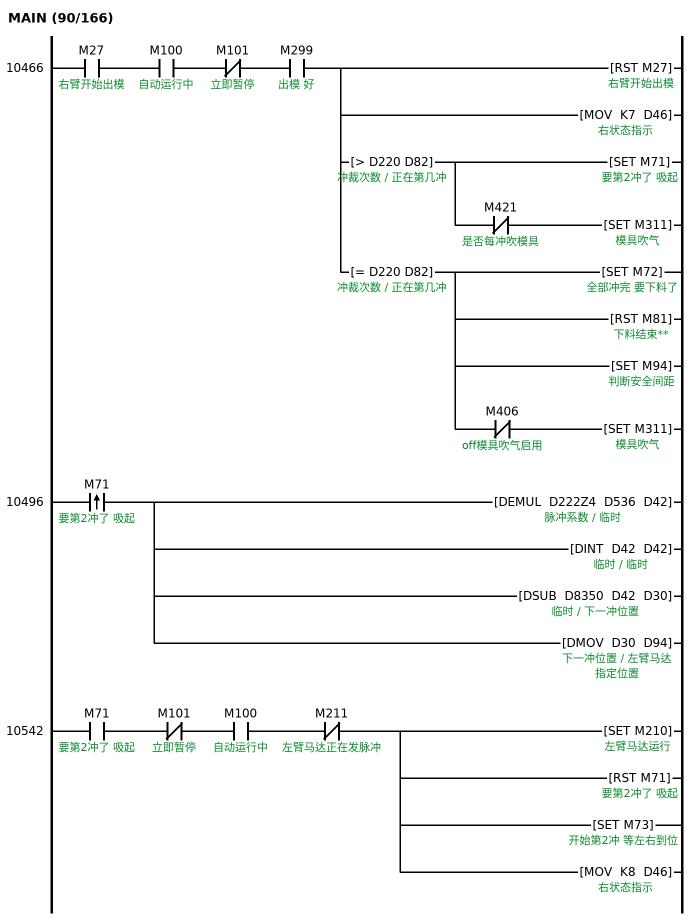
10466 LD      M27  ; 右臂开始出模
      AND     M100  ; 自动运行中
      ANI     M101  ; 立即暂停
      AND     M299  ; 出模 好
      RST     M27  ; 右臂开始出模
      MOV     K7 D46
      MPS
      AND>    D220 D82  ; 冲裁次数 / 正在第几冲
      SET     M71  ; 要第2冲了 吸起
      ANI     M421  ; 是否每冲吹模具
      SET     M311  ; 模具吹气
      MPP
      AND=    D220 D82  ; 冲裁次数 / 正在第几冲
      SET     M72  ; 全部冲完 要下料了
      RST     M81  ; 下料结束**
      SET     M94  ; 判断安全间距
      ANI     M406  ; off模具吹气启用
      SET     M311  ; 模具吹气
10496 LDP     M71  ; 要第2冲了 吸起
      DEMUL   D222Z4 D536 D42
      DINT    D42 D42
      DSUB    D8350 D42 D30  ; 下一冲位置
      DMOV    D30 D94
10542 LD      M71  ; 要第2冲了 吸起
      ANI     M101  ; 立即暂停
      AND     M100  ; 自动运行中
      ANI     M211  ; 左臂马达正在发脉冲
      SET     M210  ; 左臂马达运行
      RST     M71  ; 要第2冲了 吸起
      SET     M73  ; 开始第2冲 等左右到位
      MOV     K8 D46
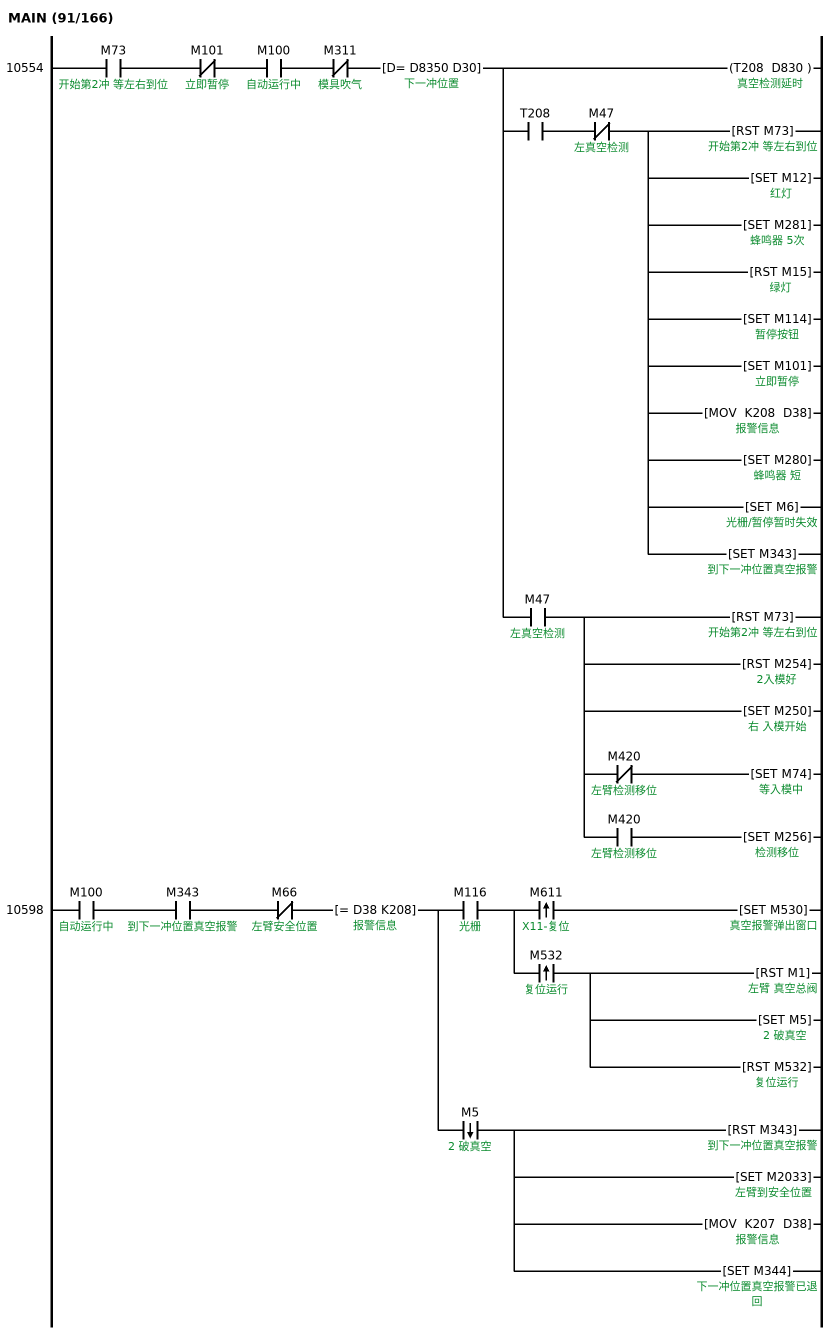
10554 LD      M73  ; 开始第2冲 等左右到位
      ANI     M101  ; 立即暂停
      AND     M100  ; 自动运行中
      ANI     M311  ; 模具吹气
      ANDD=   D8350 D30  ; 下一冲位置
      OUT     T208 D830  ; 真空检测延时
      MPS
      AND     T208
      ANI     M47  ; 左真空检测
      RST     M73  ; 开始第2冲 等左右到位
      SET     M12  ; 红灯
      SET     M281  ; 蜂鸣器 5次
      RST     M15  ; 绿灯
      SET     M114  ; 暂停按钮
      SET     M101  ; 立即暂停
      MOV     K208 D38
      SET     M280  ; 蜂鸣器 短
      SET     M6  ; 光栅/暂停暂时失效
      SET     M343  ; 到下一冲位置真空报警
      MPP
      AND     M47  ; 左真空检测
      RST     M73  ; 开始第2冲 等左右到位
      RST     M254  ; 2入模好
      SET     M250  ; 右 入模开始
      MPS
      ANI     M420  ; 左臂检测移位
      SET     M74  ; 等入模中
      MPP
      AND     M420  ; 左臂检测移位
      SET     M256  ; 检测移位
10598 LD      M100  ; 自动运行中
      AND     M343  ; 到下一冲位置真空报警
      ANI     M66  ; 左臂安全位置
      AND=    D38 K208  ; 报警信息
      MPS
      AND     M116  ; 光栅
      MPS
      ANDP    M611  ; X11-复位
      SET     M530  ; 真空报警弹出窗口
      MPP
      ANDP    M532  ; 复位运行
      RST     M1  ; 左臂 真空总阀
      SET     M5  ; 2 破真空
      RST     M532  ; 复位运行
      MPP
      ANDF    M5  ; 2 破真空
      RST     M343  ; 到下一冲位置真空报警
      SET     M2033  ; 左臂到安全位置
      MOV     K207 D38
      SET     M344  ; 下一冲位置真空报警已退回
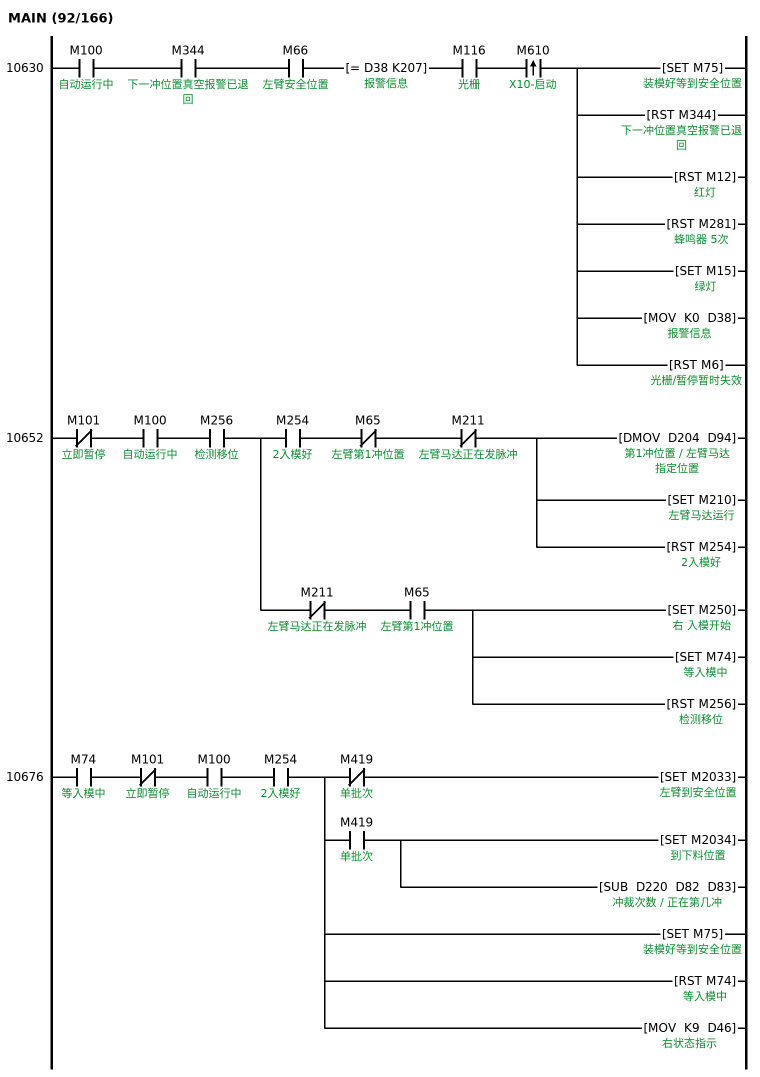
10630 LD      M100  ; 自动运行中
      AND     M344  ; 下一冲位置真空报警已退回
      AND     M66  ; 左臂安全位置
      AND=    D38 K207  ; 报警信息
      AND     M116  ; 光栅
      ANDP    M610  ; X10-启动
      SET     M75  ; 装模好等到安全位置
      RST     M344  ; 下一冲位置真空报警已退回
      RST     M12  ; 红灯
      RST     M281  ; 蜂鸣器 5次
      SET     M15  ; 绿灯
      MOV     K0 D38
      RST     M6  ; 光栅/暂停暂时失效
10652 LDI     M101  ; 立即暂停
      AND     M100  ; 自动运行中
      AND     M256  ; 检测移位
      MPS
      AND     M254  ; 2入模好
      ANI     M65  ; 左臂第1冲位置
      ANI     M211  ; 左臂马达正在发脉冲
      DMOV    D204 D94
      SET     M210  ; 左臂马达运行
      RST     M254  ; 2入模好
      MPP
      ANI     M211  ; 左臂马达正在发脉冲
      AND     M65  ; 左臂第1冲位置
      SET     M250  ; 右 入模开始
      SET     M74  ; 等入模中
      RST     M256  ; 检测移位
10676 LD      M74  ; 等入模中
      ANI     M101  ; 立即暂停
      AND     M100  ; 自动运行中
      AND     M254  ; 2入模好
      MPS
      ANI     M419  ; 单批次
      SET     M2033  ; 左臂到安全位置
      MRD
      AND     M419  ; 单批次
      SET     M2034  ; 到下料位置
      SUB     D220 D82 D83
      MPP
      SET     M75  ; 装模好等到安全位置
      RST     M74  ; 等入模中
      MOV     K9 D46
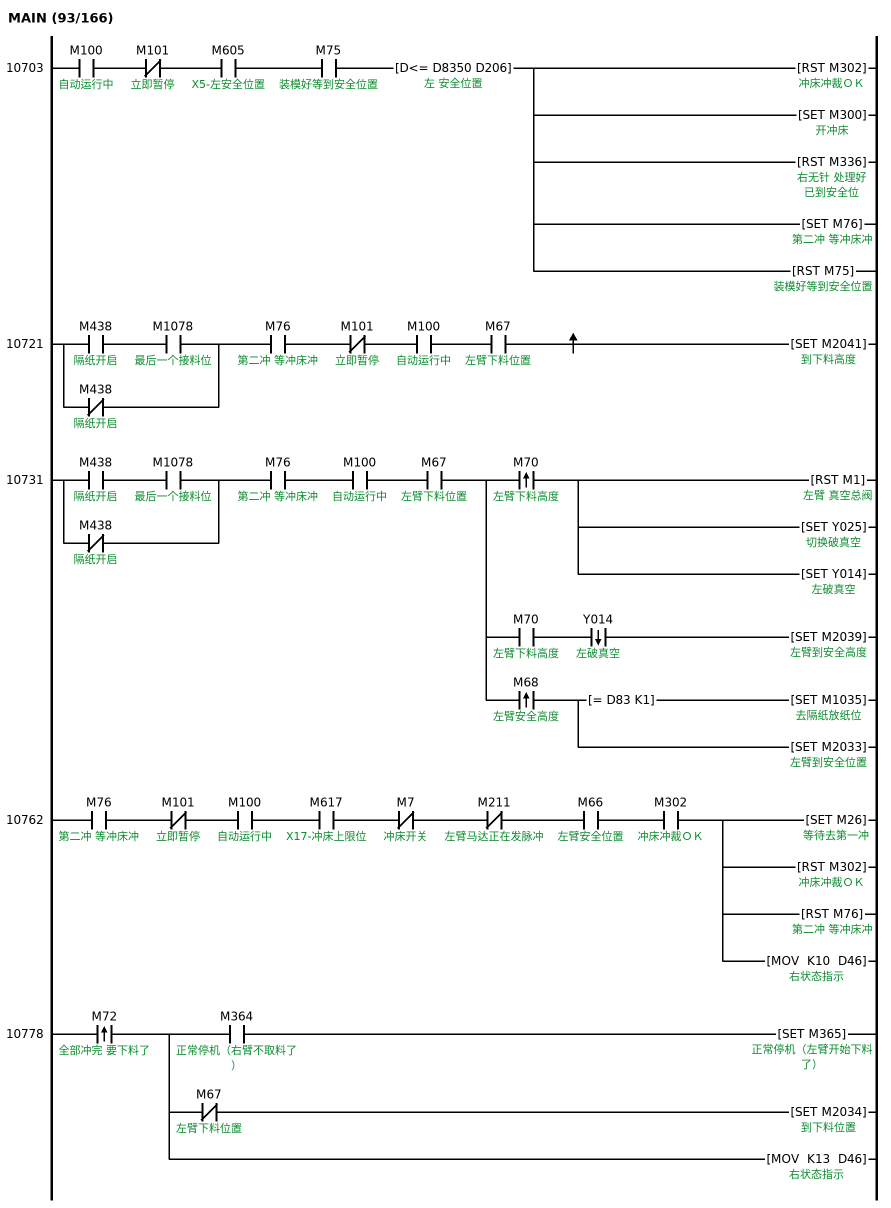
10703 LD      M100  ; 自动运行中
      ANI     M101  ; 立即暂停
      AND     M605  ; X5-左安全位置
      AND     M75  ; 装模好等到安全位置
      ANDD<=  D8350 D206  ; 左 安全位置
      RST     M302  ; 冲床冲裁ＯＫ
      SET     M300  ; 开冲床
      RST     M336  ; 右无针 处理好 已到安全位
      SET     M76  ; 第二冲 等冲床冲
      RST     M75  ; 装模好等到安全位置
10721 LD      M438  ; 隔纸开启
      AND     M1078  ; 最后一个接料位
      ORI     M438  ; 隔纸开启
      AND     M76  ; 第二冲 等冲床冲
      ANI     M101  ; 立即暂停
      AND     M100  ; 自动运行中
      AND     M67  ; 左臂下料位置
      MEP
      SET     M2041  ; 到下料高度
10731 LD      M438  ; 隔纸开启
      AND     M1078  ; 最后一个接料位
      ORI     M438  ; 隔纸开启
      AND     M76  ; 第二冲 等冲床冲
      AND     M100  ; 自动运行中
      AND     M67  ; 左臂下料位置
      MPS
      ANDP    M70  ; 左臂下料高度
      RST     M1  ; 左臂 真空总阀
      SET     Y025  ; 切换破真空
      SET     Y014  ; 左破真空
      MRD
      AND     M70  ; 左臂下料高度
      ANDF    Y014  ; 左破真空
      SET     M2039  ; 左臂到安全高度
      MPP
      ANDP    M68  ; 左臂安全高度
      MPS
      AND=    D83 K1
      SET     M1035  ; 去隔纸放纸位
      MPP
      SET     M2033  ; 左臂到安全位置
10762 LD      M76  ; 第二冲 等冲床冲
      ANI     M101  ; 立即暂停
      AND     M100  ; 自动运行中
      AND     M617  ; X17-冲床上限位
      ANI     M7  ; 冲床开关
      ANI     M211  ; 左臂马达正在发脉冲
      AND     M66  ; 左臂安全位置
      AND     M302  ; 冲床冲裁ＯＫ
      SET     M26  ; 等待去第一冲
      RST     M302  ; 冲床冲裁ＯＫ
      RST     M76  ; 第二冲 等冲床冲
      MOV     K10 D46
10778 LDP     M72  ; 全部冲完 要下料了
      MPS
      AND     M364  ; 正常停机（右臂不取料了）
      SET     M365  ; 正常停机（左臂开始下料了）
      MRD
      ANI     M67  ; 左臂下料位置
      SET     M2034  ; 到下料位置
      MPP
      MOV     K13 D46
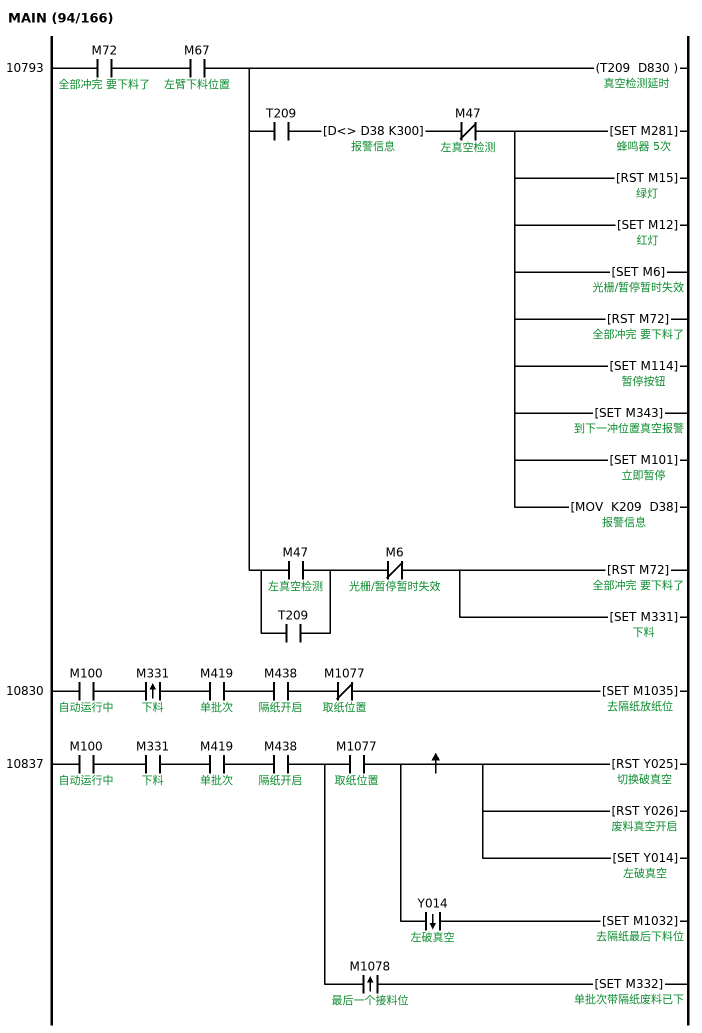
10793 LD      M72  ; 全部冲完 要下料了
      AND     M67  ; 左臂下料位置
      OUT     T209 D830  ; 真空检测延时
      MPS
      AND     T209
      ANDD<>  D38 K300  ; 报警信息
      ANI     M47  ; 左真空检测
      SET     M281  ; 蜂鸣器 5次
      RST     M15  ; 绿灯
      SET     M12  ; 红灯
      SET     M6  ; 光栅/暂停暂时失效
      RST     M72  ; 全部冲完 要下料了
      SET     M114  ; 暂停按钮
      SET     M343  ; 到下一冲位置真空报警
      SET     M101  ; 立即暂停
      MOV     K209 D38
      MPP
      LD      M47  ; 左真空检测
      OR      T209
      ANB
      ANI     M6  ; 光栅/暂停暂时失效
      RST     M72  ; 全部冲完 要下料了
      SET     M331  ; 下料
10830 LD      M100  ; 自动运行中
      ANDP    M331  ; 下料
      AND     M419  ; 单批次
      AND     M438  ; 隔纸开启
      ANI     M1077  ; 取纸位置
      SET     M1035  ; 去隔纸放纸位
10837 LD      M100  ; 自动运行中
      AND     M331  ; 下料
      AND     M419  ; 单批次
      AND     M438  ; 隔纸开启
      MPS
      AND     M1077  ; 取纸位置
      MPS
      MEP
      RST     Y025  ; 切换破真空
      RST     Y026  ; 废料真空开启
      SET     Y014  ; 左破真空
      MPP
      ANDF    Y014  ; 左破真空
      SET     M1032  ; 去隔纸最后下料位
      MPP
      ANDP    M1078  ; 最后一个接料位
      SET     M332  ; 单批次带隔纸废料已下
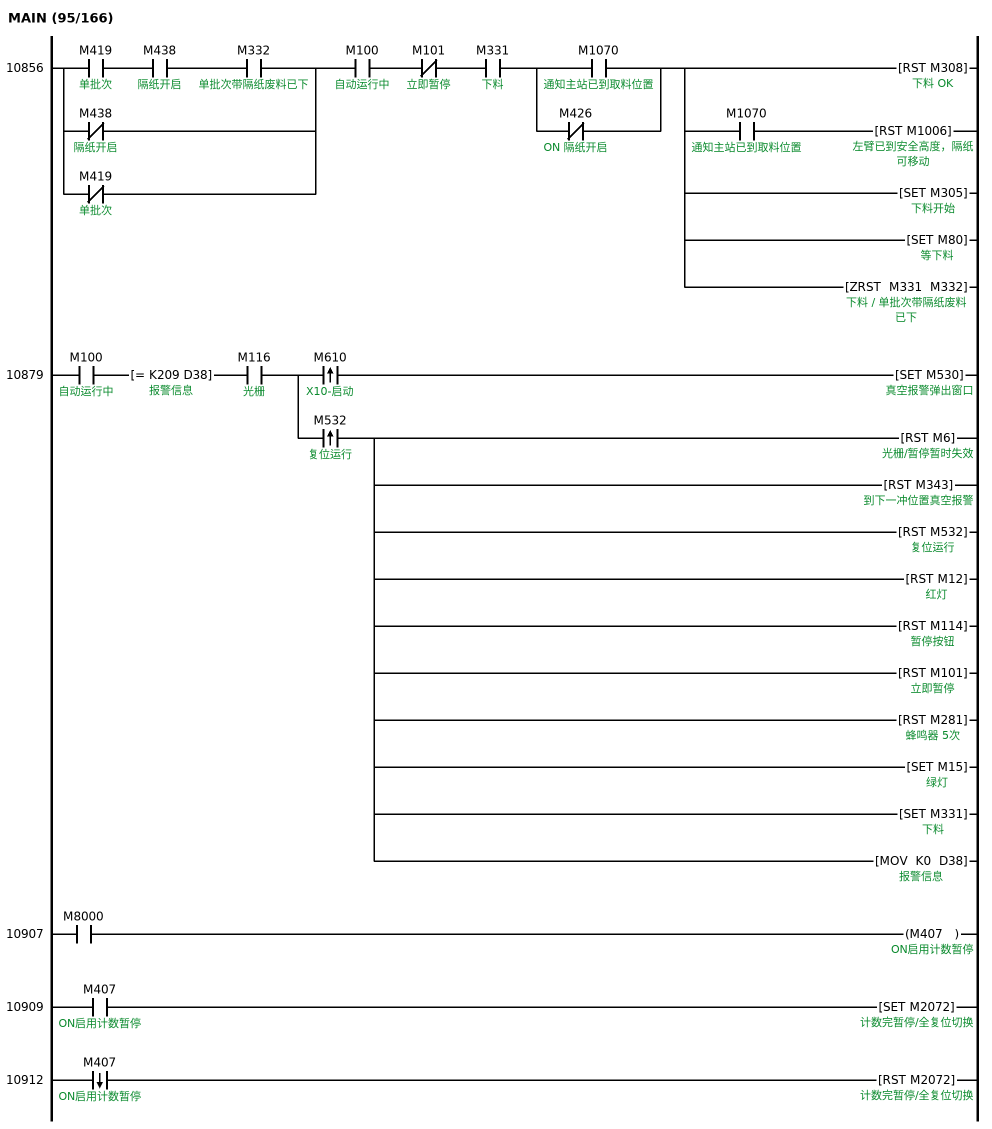
10856 LD      M419  ; 单批次
      AND     M438  ; 隔纸开启
      AND     M332  ; 单批次带隔纸废料已下
      ORI     M438  ; 隔纸开启
      ORI     M419  ; 单批次
      AND     M100  ; 自动运行中
      ANI     M101  ; 立即暂停
      AND     M331  ; 下料
      LD      M1070  ; 通知主站已到取料位置
      ORI     M426  ; ON 隔纸开启
      ANB
      RST     M308  ; 下料 OK
      MPS
      AND     M1070  ; 通知主站已到取料位置
      RST     M1006  ; 左臂已到安全高度，隔纸可移动
      MPP
      SET     M305  ; 下料开始
      SET     M80  ; 等下料
      ZRST    M331 M332
10879 LD      M100  ; 自动运行中
      AND=    K209 D38  ; 报警信息
      AND     M116  ; 光栅
      MPS
      ANDP    M610  ; X10-启动
      SET     M530  ; 真空报警弹出窗口
      MPP
      ANDP    M532  ; 复位运行
      RST     M6  ; 光栅/暂停暂时失效
      RST     M343  ; 到下一冲位置真空报警
      RST     M532  ; 复位运行
      RST     M12  ; 红灯
      RST     M114  ; 暂停按钮
      RST     M101  ; 立即暂停
      RST     M281  ; 蜂鸣器 5次
      SET     M15  ; 绿灯
      SET     M331  ; 下料
      MOV     K0 D38
10907 LD      M8000
      OUT     M407  ; ON启用计数暂停
10909 LD      M407  ; ON启用计数暂停
      SET     M2072  ; 计数完暂停/全复位切换
10912 LDF     M407  ; ON启用计数暂停
      RST     M2072  ; 计数完暂停/全复位切换
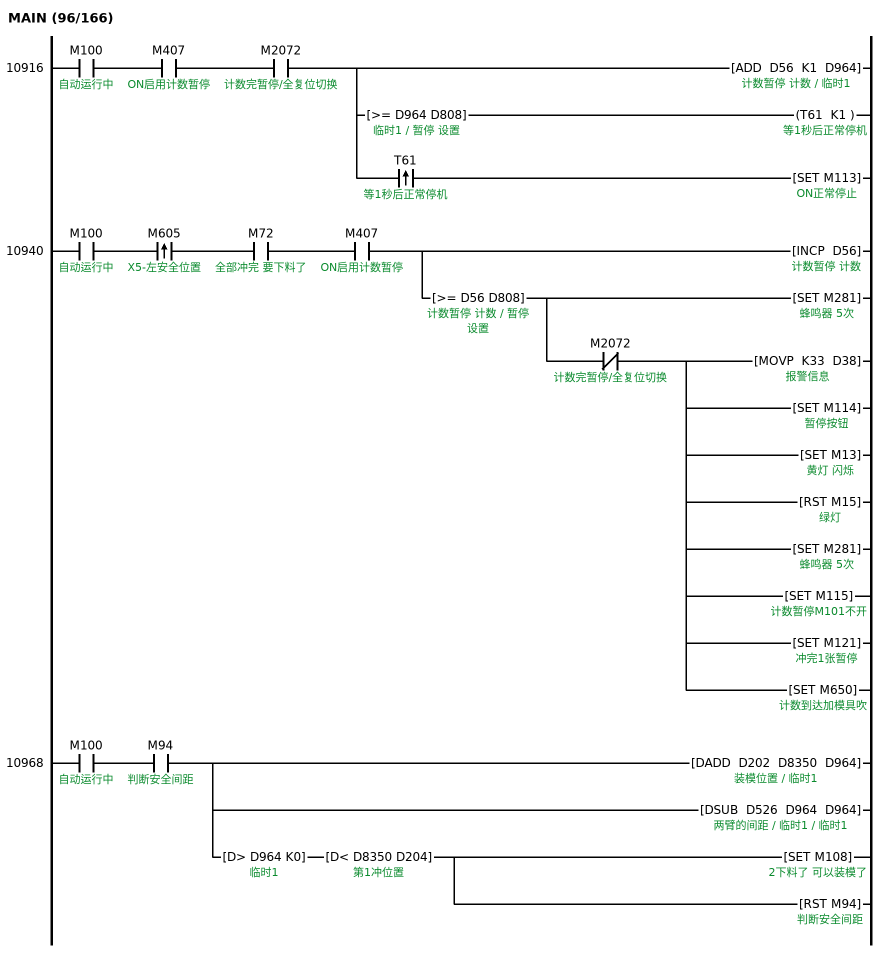
10916 LD      M100  ; 自动运行中
      AND     M407  ; ON启用计数暂停
      AND     M2072  ; 计数完暂停/全复位切换
      ADD     D56 K1 D964
      MPS
      AND>=   D964 D808  ; 临时1 / 暂停 设置
      OUT     T61 K1  ; 等1秒后正常停机
      MPP
      ANDP    T61  ; 等1秒后正常停机
      SET     M113  ; ON正常停止
10940 LD      M100  ; 自动运行中
      ANDP    M605  ; X5-左安全位置
      AND     M72  ; 全部冲完 要下料了
      AND     M407  ; ON启用计数暂停
      INCP    D56
      AND>=   D56 D808  ; 计数暂停 计数 / 暂停 设置
      SET     M281  ; 蜂鸣器 5次
      ANI     M2072  ; 计数完暂停/全复位切换
      MOVP    K33 D38
      SET     M114  ; 暂停按钮
      SET     M13  ; 黄灯 闪烁
      RST     M15  ; 绿灯
      SET     M281  ; 蜂鸣器 5次
      SET     M115  ; 计数暂停M101不开
      SET     M121  ; 冲完1张暂停
      SET     M650  ; 计数到达加模具吹
10968 LD      M100  ; 自动运行中
      AND     M94  ; 判断安全间距
      DADD    D202 D8350 D964
      DSUB    D526 D964 D964
      ANDD>   D964 K0  ; 临时1
      ANDD<   D8350 D204  ; 第1冲位置
      SET     M108  ; 2下料了 可以装模了
      RST     M94  ; 判断安全间距
